Staubli VAL3: shiftRight.pgx

public program shiftRight(string& x_sBinary, num x_nPos)
  local bool l_bIsBinary
  local string l_sBinary
  local num l_nIndex
begin

  l_bIsBinary=false
  call isBinary(x_sBinary, l_bIsBinary)
  l_sBinary = x_sBinary

  if l_bIsBinary
    for l_nIndex=0 to x_nPos-1
      l_sBinary = "0"+l_sBinary
    endFor
    x_sBinary=left(l_sBinary, len(x_sBinary))
  else
    logMsg("Binary->shiftLeft: wrong input format")
  endIf

end
